// TIA Portal V20 export
VAR_GLOBAL   // PLC tag table "PLC_Functional_Test"
   Button_Start_Approve AT %I0.0 : Bool;
   Digital_Input_1 AT %I0.1 : Bool;
   Digital_Input_2 AT %I0.2 : Bool;
   Digital_Input_3 AT %I0.3 : Bool;
   Digital_Input_4 AT %I0.4 : Bool;
   Digital_Input_5 AT %I0.5 : Bool;
   Current_Transducer AT %IW64 : Int;
   Voltage_Transducer AT %IW66 : Int;
   Button_Light AT %Q0.0 : Bool;
   Light_Fail_Test AT %Q0.1 : Bool;
   Light_Approve_Test AT %Q0.2 : Bool;
   Digital_Output_3 AT %Q0.3 : Bool;
   Clock_Byte AT %MB0 : Byte;
   Clock_10Hz AT %M0.0 : Bool;
   Clock_5Hz AT %M0.1 : Bool;
   "Clock_2.5Hz" AT %M0.2 : Bool;
   Clock_2Hz AT %M0.3 : Bool;
   "Clock_1.25Hz" AT %M0.4 : Bool;
   Clock_1Hz AT %M0.5 : Bool;
   "Clock_0.625Hz" AT %M0.6 : Bool;
   "Clock_0.5Hz" AT %M0.7 : Bool;
   System_Byte AT %MB1 : Byte;
   FirstScan AT %M1.0 : Bool;
   DiagStatusUpdate AT %M1.1 : Bool;
   AlwaysTRUE AT %M1.2 : Bool;
   AlwaysFALSE AT %M1.3 : Bool;
END_VAR
